(*			
	RafalOS
	Rafał Osajda		19.11.2025		TC 4024.66
	Domyślne przygotowanie danych dla ekranu
*)
FUNCTION_BLOCK FB_MCHMIPrepareDataForScreen EXTENDS FB_BaseComponent_HMI IMPLEMENTS ITF_MCHMIPrepareScreen_Init
VAR
	//itf do lacznika machinecontrol
	//strulture danych 
	itfExtendedDisplay			: ITF_MCHMIDisplayExtension;
END_VAR

(*			
	RafalOS
	Rafał Osajda		19.11.2025		TC 4024.66
	Czyści danych przy zmienia ramki po poprzedniej ramce
*)
METHOD PUBLIC ClearAfterScreen : BOOL
VAR_INPUT
END_VAR
IF (THIS^.itfExtendedDisplay <> 0) THEN
	THIS^.itfExtendedDisplay.ExtendedClearAfterScreen ();
END_IF
END_METHOD

METHOD PUBLIC LinkDataHMI_00_01 : BOOL
VAR_INPUT
	refstData				: REFERENCE TO ST_MCHMIPrepareScreen_00_01;
END_VAR
END_METHOD

METHOD PUBLIC LinkDataHMI_00_02 : BOOL
VAR_INPUT
	refstData				: REFERENCE TO ST_MCHMIPrepareScreen_00_02;
END_VAR
END_METHOD

METHOD PUBLIC LinkDataHMI_00_03 : BOOL
VAR_INPUT
	refstData				: REFERENCE TO ST_MCHMIPrepareScreen_00_03;
END_VAR
END_METHOD

METHOD PUBLIC LinkDataHMI_00_04 : BOOL
VAR_INPUT
	refstData				: REFERENCE TO ST_MCHMIPrepareScreen_00_04;
END_VAR
END_METHOD

METHOD PUBLIC LinkDataHMI_00_05 : BOOL
VAR_INPUT
	refstData				: REFERENCE TO ST_MCHMIPrepareScreen_00_05;
END_VAR
END_METHOD

METHOD PUBLIC LinkDataHMI_01_XX : BOOL
VAR_INPUT
	refstData				: REFERENCE TO ST_MCHMIPrepareScreen_01_XX;
END_VAR
END_METHOD

METHOD PUBLIC LinkDataHMI_02_XX : BOOL
VAR_INPUT
	refstData				: REFERENCE TO ST_MCHMIPrepareScreen_02_XX;
END_VAR
END_METHOD

METHOD PUBLIC LinkDataHMI_03_XX : BOOL
VAR_INPUT
	refstData				: REFERENCE TO ST_MCHMIPrepareScreen_03_XX;
END_VAR
END_METHOD

METHOD PUBLIC LinkDataHMI_04_XX : BOOL
VAR_INPUT
	refstData				: REFERENCE TO ST_MCHMIPrepareScreen_04_XX;
END_VAR
END_METHOD

METHOD PUBLIC LinkDataHMI_05_XX : BOOL
VAR_INPUT
	refstData				: REFERENCE TO ST_MCHMIPrepareScreen_05_XX;
END_VAR
END_METHOD

METHOD PUBLIC LinkDataHMI_06_XX : BOOL
VAR_INPUT
	refstData				: REFERENCE TO ST_MCHMIPrepareScreen_06_XX;
END_VAR
END_METHOD

METHOD PUBLIC LinkDataHMI_07_XX : BOOL
VAR_INPUT
	refstData				: REFERENCE TO ST_MCHMIPrepareScreen_07_XX;
END_VAR
END_METHOD

METHOD PUBLIC LinkExtensionDisplay : BOOL
VAR_INPUT
	fbExtendedDisplay			: ITF_MCHMIDisplayExtension;
END_VAR
THIS^.itfExtendedDisplay := fbExtendedDisplay;
END_METHOD

(*			
	RafalOS
	Rafał Osajda		14.11.2025		TC 4024.66
	Metoda przygotowywania danych dla HMI 
	W niej odbywa się odpytywanie właściego elementu przez łącznik
*)
METHOD PUBLIC PrepareDataForHMI : BOOL
VAR_INPUT
END_VAR
IF (THIS^.itfExtendedDisplay <> 0) THEN
	THIS^.itfExtendedDisplay.ExtendedPrepareDataForHMI ();
END_IF
END_METHOD

(*			
	RafalOS
	Rafał Osajda		19.11.2025		TC 4024.66
	Przygotowanie ramki pood tamke do wyświetlenia - tylko przygotowanie a nie przygotowanie danych do wyświetlenia
*)
METHOD PUBLIC PrepareForScreen : BOOL
VAR_INPUT
END_VAR
IF (THIS^.itfExtendedDisplay <> 0) THEN
	THIS^.itfExtendedDisplay.ExtendedPrepareForScreen ();
END_IF
END_METHOD

END_FUNCTION_BLOCK

(* stored: Version 1.1.0.1
   POU FB_MCHMIPrepareDataForScreen: Id {3050d0c5-d80e-0889-00e3-5f0104bdd004}, SpecialFunc None
   Folder ITF_Init: Id {8b968d7c-09bf-07b6-1c78-8a1436fa4012}
   Folder ITF_PDFS: Id {5ed5ea20-8c25-034d-2252-9059bf81fcb7}
   Method ClearAfterScreen: Id {9877e0d9-8678-0ae8-355c-333615fe32d2}
   Method LinkDataHMI_00_01: Id {02b6a1d7-d2e7-0d96-1a06-125016d837fd}
   Method LinkDataHMI_00_02: Id {1845f68e-bb67-0bb0-0014-7d4a64071beb}
   Method LinkDataHMI_00_03: Id {8ebbb9ec-ac0d-0603-2b3d-1d6587257fa3}
   Method LinkDataHMI_00_04: Id {850e4e53-e593-068e-3d0b-357841e59ebc}
   Method LinkDataHMI_00_05: Id {862d07cc-c025-0f7d-0d4e-5a2f317ce50a}
   Method LinkDataHMI_01_XX: Id {ea4ca59d-69b8-0d18-3dc0-015aa5af68ee}
   Method LinkDataHMI_02_XX: Id {a1128685-79de-030f-39b5-2f5a3cd092bf}
   Method LinkDataHMI_03_XX: Id {4319d5c0-d837-06e9-0760-3018e67c124c}
   Method LinkDataHMI_04_XX: Id {3c1def7f-03cf-027c-0bcf-e1bc0ca53b26}
   Method LinkDataHMI_05_XX: Id {e200060d-69b9-0ae8-0d21-dafbb767bf8f}
   Method LinkDataHMI_06_XX: Id {565b628b-139c-0646-26c5-ddaf3aef254b}
   Method LinkDataHMI_07_XX: Id {5849f20e-11ca-06a2-278b-1cb6412c0501}
   Method LinkExtensionDisplay: Id {f5e43dfa-4e83-0f5f-10aa-f7a9025acd9b}
   Method PrepareDataForHMI: Id {bc2b143f-e4a1-0155-38ef-904b1a2f8b08}
   Method PrepareForScreen: Id {28b2ca1f-8b84-0c44-1ac0-89ac26d6625e} *)
